FUNCTION_BLOCK "FB_Dispatch_Point_T"
TITLE = %version: 5.09 % %Commit:  c3808b61 % CN: 50
{ S7_Optimized_Access := 'FALSE' }
FAMILY : Tubtrax
VERSION : 0.0

BEGIN

NETWORK
TITLE = BA: Search for item on Dispatch Point
      NOP 0;
      L #t_Fnd_Num_Items_Leading;
AA01: L 0;
      >I;
      = #t_Carrier_Found;

NETWORK
TITLE = BB: Initialize values when new carrier found
      NOP 0;
      L #t_TIC;
      L 0;
      >I;
bb01: JCN BB99;

// Determine if LIC present
      CALL "FC_Read_Int_Record"
      (  i_Record_Number             := #t_LNK ,
         i_P_INT_Record              := "DB_UDT_LNK_Record".LIC ,
         i_DB                        := "DB_LNK_List" ,
         i_DB_Event_Num              := #t_DB_Event_Section ,
         o_INT                       := #s_LIC
      );

// Determine if carrier is loaded
      L #s_LIC;
      L 0;
      >I;
      AN #t_Tub_Unknown;
      A #t_Tub_Loaded;
      S #s_Carrier_Loaded;

BB99:      NOP 0;

NETWORK
TITLE = BC: Send package report when arriving
      NOP 0;

// If loaded carrier arriving
      A #s_FP_Carrier_Found;
      A #s_Carrier_Loaded;
      JCN BC99;

      CALL "FC_Read_Int_Record"
      (  i_Record_Number             := #t_LNK ,
         i_P_INT_Record              := "DB_UDT_LNK_Record".ECS ,
         i_DB                        := "DB_LNK_List" ,
         i_DB_Event_Num              := #t_DB_Event_Section ,
         o_INT                       := #t_ECS
      );

// 1211 = Package Report (Arrived)
      CALL "FC_Write_Event"
      (  i_Message_ID                := 1211 ,
         i_Event_value               := #t_LNK ,
         i_DB_Event_Num              := #t_DB_Event_Section ,
         o_Return_Value              := #t_Not_Used_Int
      );

BC99:      NOP 0;

NETWORK
TITLE = CA: Check and set destination
//If a Bag has the Dispatch Point as destination this network will search a
//valid destination that is available and that wasn't used recently, if any of
//these conditions isn't verified this network will check the same conditions for
//the next destination.
      NOP 0;

      A #t_Carrier_Found;
      A #s_Carrier_Loaded;
      A(;
      L #s_Available_Destination;
      L 0;
      ==I;
      );
      JCN CA99;

// If destination bigger than zero
CA001:      L W[ AR1, P#0.0];
      L 0;
      >I;
      JCN CA02;

// AND destination available
      A[ AR1, P#2.0];
      JCN CA02;

// AND NOT used recently
      AN[ AR2, P#0.0];
      JCN CA02;

// Copy Destination in result
      L W[ AR1, P#0.0];
      T #t_Destination_Found;

// Set entry as used
      SET;
      S[ AR2, P#0.0];

      JU CA03;

// If destination equal or smaller than zero OR not available, checks next destination and availability
CA02:      L P#4.0;
      +AR1;

      L P#0.1;
      +AR2;

// Increment 1 to the loop counter until a maximum of 15 destinations
      L #t_Loop_Counter;
      L 1;
      +I;
      T #t_Loop_Counter;

      L #t_Loop_Counter;
      L 15;
      >I;
      JCN CA01;

// Restore AR content
CA3:      L #t_AR1_Backup;
      LAR1;
      L #t_AR2_Backup;
      LAR2;

      L #t_Destination_Found;
      T #s_Available_Destination;

CA99:      NOP 0;

NETWORK
TITLE = DA: Reset 'used' property
//When there is no 'available' and not 'used' station, reset 'used' indicator of
//all stations
DA00: NOP 0;

// Carrier on Dispatch Point AND destinations not available
DA01: A #t_Carrier_Found;
      A #s_Carrier_Loaded;
      A(;
      L #s_Available_Destination;
      L 0;
      ==I;
      );
      JCN DA99;

// Preset Loop counter
DA02: L 1;
      T #t_Loop_Counter;

// Backup AR content
DA03: TAR1;
      T #t_AR1_Backup;
      TAR2;
      T #t_AR2_Backup;

// Load start position AR1 and AR2
      LAR1 P##i_Destination_01;
      LAR2 P##s_Dest_01_Used;

// If destination bigger than zero
DA02: L W[ AR1, P#0.0];
      L 0;
      >I;
      JCN DA02;

// Reset destination used
      SET;
      R[ AR2, P#0.0];

// If destination equal or smaller than zero OR not available, checks next destination and availability
DA04: L P#4.0;
      +AR1;

      L P#0.1;
      +AR2;

// Increment 1 to the loop counter until a maximum of 15 destinations
DA04: L #t_Loop_Counter;
      L 1;
      +I;
      T #t_Loop_Counter;

      L #t_Loop_Counter;
      L 15;
      >I;
      JCN DA01;

      NOP 0;

// Restore AR content
      L #t_AR1_Backup;
      LAR1;
      L #t_AR2_Backup;
      LAR2;

DA99:      NOP 0;

NETWORK
TITLE = EA: Assign carrier to a destination
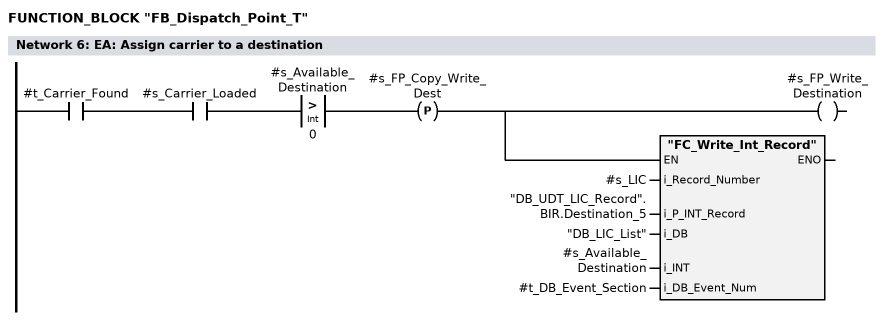
      NOP 0;

      A #t_Carrier_Found;
      A #s_Carrier_Loaded;
      A(;
      L #s_Available_Destination;
      L 0;
      >I;
      );
      FP #s_FP_Copy_Write_Dest;
      = #s_FP_Write_Destination;
      JCN EA99;

// Write destination of the assigned destination in the LIC record
      CALL "FC_Write_Int_Record"
      (  i_Record_Number             := #s_LIC ,
         i_P_INT_Record              := "DB_UDT_LIC_Record".BIR.Destination_5 ,
         i_DB                        := "DB_LIC_List" ,
         i_INT                       := #s_Available_Destination ,
         i_DB_Event_Num              := #t_DB_Event_Section
      );

EA99:      NOP 0;

NETWORK
TITLE = EB: Send tracking report when leaving
      NOP 0;

// Determine when loaded carrier is assigned to OPZ
      A #s_FP_Write_Destination;
      JCN EB99;

      L #t_LNK;
      L 0;
      >I;
      JCN EB99;

// Read TIC number from LNK list
      CALL "FC_Read_Int_Record"
      (  i_Record_Number             := #t_LNK ,
         i_P_INT_Record              := "DB_UDT_LNK_Record".TIC ,
         i_DB                        := "DB_LNK_List" ,
         i_DB_Event_Num              := #t_DB_Event_Section ,
         o_INT                       := #t_TIC
      );

// Check if TIC number is valid
      L #t_TIC;
      L 0;
      >I;
      JCN EB99;

// Read LIC number from LNK list
      CALL "FC_Read_Int_Record"
      (  i_Record_Number             := #t_LNK ,
         i_P_INT_Record              := "DB_UDT_LNK_Record".LIC ,
         i_DB                        := "DB_LNK_List" ,
         i_DB_Event_Num              := #t_DB_Event_Section ,
         o_INT                       := #t_LIC
      );

// Read report route number from LNK list
      CALL "FC_Read_Int_Record"
      (  i_Record_Number             := #t_LNK ,
         i_P_INT_Record              := "DB_UDT_LNK_Record".Rep_Route ,
         i_DB                        := "DB_LNK_List" ,
         i_DB_Event_Num              := #t_DB_Event_Section ,
         o_INT                       := #t_Rep_Route_Record
      );

// Clear LNK from report route record
      L #t_Rep_Route_Record;
      L 0;
      >I;
      JCN EB01;

      CALL "FC_Write_Int_Record"
      (  i_Record_Number             := #t_Rep_Route_Record ,
         i_P_INT_Record              := "DB_UDT_Route_Record".LNK ,
         i_DB                        := "DB_Route_List" ,
         i_INT                       := 0 ,
         i_DB_Event_Num              := #t_DB_Event_Section
      );

// Clear report route record from LNK
EB01:      CALL "FC_Write_Int_Record"
      (  i_Record_Number             := #t_LNK ,
         i_P_INT_Record              := "DB_UDT_LNK_Record".Rep_Route ,
         i_DB                        := "DB_LNK_List" ,
         i_INT                       := 0 ,
         i_DB_Event_Num              := #t_DB_Event_Section
      );

// Generate new route record
      CALL "FC_Generator_LNK"
      (  i_LNK                       := #t_LNK ,
         i_DB_List                   := #t_DB_Route_List_Num ,
         i_Default_Record            := -1 ,
         i_DB_Event_Num              := #t_DB_Event_Section ,
         o_LNK                       := #t_Rep_Route_Record
      );

// Read report route number from LNK list
      CALL "FC_Read_Int_Record"
      (  i_Record_Number             := #t_LNK ,
         i_P_INT_Record              := "DB_UDT_LNK_Record".Rep_Route ,
         i_DB                        := "DB_LNK_List" ,
         i_DB_Event_Num              := #t_DB_Event_Section ,
         o_INT                       := #t_Rep_Route_Record
      );

// Copy BIR to report route record
      CALL "FC_Read_ANY_Record"
      (  i_Record_Number             := #t_LIC ,
         i_ANY_Data_Record           := "DB_UDT_LIC_Record".BIR ,
         i_ANY_Data                  := "DB_Outgoing_Msgs".TrackingReport.Body.BIR ,
         i_DB                        := "DB_LIC_List" ,
         i_DB_Event_Num              := #t_DB_Event_Section
      );

      CALL "FC_Write_ANY_Record"
      (  i_Record_Number             := #t_Rep_Route_Record ,
         i_ANY_Data_Record           := "DB_UDT_Route_Record".BIR ,
         i_ANY_Data                  := "DB_Outgoing_Msgs".TrackingReport.Body.BIR ,
         i_DB                        := "DB_Route_List" ,
         i_DB_Event_Num              := #t_DB_Event_Section
      );

// Copy LIC number to report route record
      CALL "FC_Write_Int_Record"
      (  i_Record_Number             := #t_Rep_Route_Record ,
         i_P_INT_Record              := "DB_UDT_Route_Record".LIC ,
         i_DB                        := "DB_Route_List" ,
         i_INT                       := #t_LIC ,
         i_DB_Event_Num              := #t_DB_Event_Section
      );

// 1201 = Tracking report
      CALL "FC_Write_Event"
      (  i_Message_ID                := 1201 ,
         i_Event_value               := #t_LNK ,
         i_DB_Event_Num              := #t_DB_Event_Section ,
         o_Return_Value              := #t_Not_Used_Int
      );

EB99:      NOP 0;

NETWORK
TITLE = EC: Move carrier from upstream buffer to downstream buffer
//At the route segment transition the data has to be moved to the correct carrier
//buffer DB.
      NOP 0;

// Move carrier to route segment buffer DB
      CALL #s_FB_Rte_Seg_FIFO_T
      (  i_CFG_Position_Node         := #i_CFG_Position_Node ,
         i_CFG_Area_HO_Dwnstr        := FALSE ,
         i_DB_PLT_Node               := #i_DB_PLT ,
         i_DB_RS_Upstr               := #i_DB_RS_Upstr ,
         i_DB_RS_Dwnstr              := #i_DB_RS_Dwnstr ,
         i_DB_Event                  := "DB_Event_Section"
      );

NETWORK
TITLE = FA: Reset/Set Carrier assigned
      NOP 0;

// Determine if a new destination is selected
      L #s_Available_Destination;
      L 0;
      >I;
      JCN FA01;

// Set carrier assigned when carrier is assigned AND item at handover
      A(;
      L #s_Available_Destination;
      L #i_Destination_01;
      ==I;
      );
      A #t_Section_Item_At_HO;
      S #o_Carrier_Assigned_01;

FA01:      NOP 0;

      A #i_Dest_15_Available;
      FP #s_FP_Dest_15_Avail;
      R #o_Carrier_Assigned_15;

END_FUNCTION_BLOCK
